FUNCTION_BLOCK FB_EncoderScalingNC_TestDouble IMPLEMENTS I_EncoderScaling

PROPERTY EncoderCount : UDINT
GET
END_GET
END_PROPERTY

METHOD EncoderScaling : UDINT
END_METHOD

END_FUNCTION_BLOCK

(* stored: Version 1.1.0.1
   POU FB_EncoderScalingNC_TestDouble: Id {3f8ce75b-8ee3-4620-85ff-fbc59d6ed483}, SpecialFunc None
   Property EncoderCount: Id {58ecbc98-356a-4ee2-b9ec-aa8c2efc18bc}
   Get Get: Id {a01045c9-3059-4366-aa1d-36f7b5ffd107}
   Method EncoderScaling: Id {3ac4197f-c191-40c5-8820-fb0a9b2c5a9d} *)
